// Mitsubishi GX Works2 project: 241108_PLC_PRACTICE2   PLC: Q02U

PROGRAM MAIN
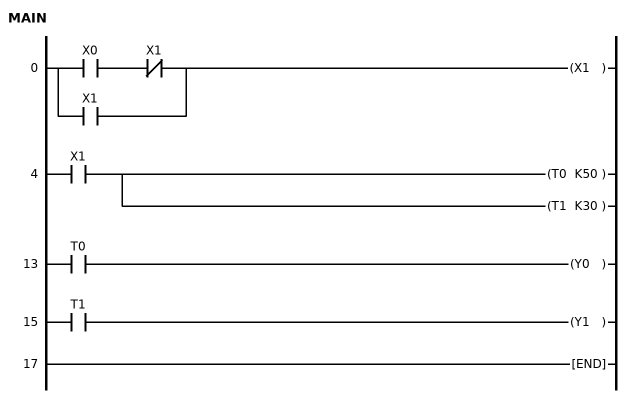
0     LD      X0
      ANI     X1
      OR      X1
      OUT     X1
4     LD      X1
      OUT     T0 K50
      OUT     T1 K30
13    LD      T0
      OUT     Y0
15    LD      T1
      OUT     Y1
17    END
END_PROGRAM
